{attribute 'qualified_only'}
VAR_GLOBAL
	FbPersistentManager : FB_PersistentDataManager ;
END_VAR

(* stored: Version 1.1.0.1, ProductVersion 3.1.4024.2
   GVL DataManager: Id {a7a689c2-2421-4e24-91c7-6cb14ea8f288} *)
